FUNCTION_BLOCK PLCopenCallGroup IMPLEMENTS IPLCopenCall
VAR_INPUT
END_VAR
VAR_OUTPUT
END_VAR
VAR
    _callGroup : PLCopenCallGroupType;
END_VAR

// Copyright (c) 2024 Loupe (https://loupe.team), provided under the MIT License.

METHOD Aborted : BOOL
// Copyright (c) 2024 Loupe (https://loupe.team), provided under the MIT License.

_callGroup._syncAbort := TRUE;
END_METHOD

METHOD PRIVATE CheckStatus : BOOL
VAR
    _commandIndex : INT;
    _anyAbort : BOOL;
    _anyBusy : BOOL;
    _anyError : BOOL;
END_VAR
// Copyright (c) 2024 Loupe (https://loupe.team), provided under the MIT License.

//If it's not in the list
FOR _commandIndex := 0 TO GVLTcCommando.MAX_RELATED_GROUPS DO
    IF _callGroup._commands[_commandIndex].Command <> 0 THEN
        _callGroup._commands[_commandIndex]();

        IF _callGroup._commands[_commandIndex].CommandAborted THEN
            _anyAbort := TRUE;
        ELSIF _callGroup._commands[_commandIndex].Error THEN
            _anyError := TRUE;
        ELSIF _callGroup._commands[_commandIndex].Busy THEN
            _anyBusy := TRUE;
        ELSE
            _callGroup._commands[_commandIndex].Command := 0;
        END_IF
    END_IF
END_FOR

_callGroup._isError := FALSE;
_callGroup._isAbort := FALSE;
_callGroup._isDone := FALSE;

IF _anyError OR _callGroup._syncError THEN
    _callGroup._isError := TRUE;
ELSIF _anyAbort OR _callGroup._syncAbort THEN
    _callGroup._isAbort := TRUE;
ELSIF NOT _anyBusy THEN
    _callGroup._isDone := TRUE;
END_IF
END_METHOD

METHOD Errored : BOOL
VAR_INPUT
    ID : INT;
END_VAR
// Copyright (c) 2024 Loupe (https://loupe.team), provided under the MIT License.

_callGroup._syncError := TRUE;
END_METHOD

METHOD Finished : BOOL
// Copyright (c) 2024 Loupe (https://loupe.team), provided under the MIT License.

_callGroup._syncDone := TRUE;
END_METHOD

PROPERTY IsAbort : BOOL
GET
// Copyright (c) 2024 Loupe (https://loupe.team), provided under the MIT License.

CheckStatus();
IsAbort := _callGroup._isAbort;
END_GET
END_PROPERTY

PROPERTY IsDone : BOOL
GET
// Copyright (c) 2024 Loupe (https://loupe.team), provided under the MIT License.

CheckStatus();

//Check if we are done
IsDone := _callGroup._isDone;
END_GET
END_PROPERTY

PROPERTY IsError : BOOL
GET
// Copyright (c) 2024 Loupe (https://loupe.team), provided under the MIT License.

CheckStatus();

IsError := _callGroup._isError;
END_GET
END_PROPERTY

{warning 'add method implementation '}
METHOD PLCopenCall : PLCopenStatusBase
VAR_INPUT
    Command : IPLCopenCommand;
END_VAR
// Copyright (c) 2024 Loupe (https://loupe.team), provided under the MIT License.
END_METHOD

METHOD ResetCommands : BOOL
VAR
    _commandIndex : INT;
END_VAR
// Copyright (c) 2024 Loupe (https://loupe.team), provided under the MIT License.

//If it's not in the list
FOR _commandIndex := 0 TO GVLTcCommando.MAX_RELATED_GROUPS DO
    _callGroup._commands[_commandIndex].Clear();
END_FOR
END_METHOD

METHOD Start : BOOL
VAR_INPUT
    Command : IPLCopenCommand;
END_VAR
VAR
    _commandIndex : INT;
END_VAR
// Copyright (c) 2024 Loupe (https://loupe.team), provided under the MIT License.

// Check if it's already in the list
FOR _commandIndex := 0 TO GVLTcCommando.MAX_RELATED_GROUPS DO
    IF _callGroup._commands[_commandIndex].Command = Command THEN
        _callGroup._commands[_commandIndex].Exec(Command);
        Start := TRUE;
        RETURN;
    END_IF
END_FOR

// If it's not in the list
FOR _commandIndex := 0 TO GVLTcCommando.MAX_RELATED_GROUPS DO
    IF _callGroup._commands[_commandIndex].Command = 0 THEN
        _callGroup._commands[_commandIndex].Exec(Command);
        Start := TRUE;
        RETURN;
    END_IF
END_FOR

Start := FALSE;

//TODO: All out of commands.. Throw an error
END_METHOD

END_FUNCTION_BLOCK

(* stored: Version 1.1.0.1
   POU PLCopenCallGroup: Id {cba9c738-238a-4f8b-b4d1-3486de669f1d}, SpecialFunc None
   Folder PLCopenCaller: Id {b4b03af3-7533-4298-bf9d-09121bd9eae9}
   Method Aborted: Id {88516a3e-7cba-4182-ba66-c0dd75064666}
   Method CheckStatus: Id {69b5b758-9323-4002-906a-f59304b6dbf8}
   Method Errored: Id {2a110df0-07b9-4922-ba19-6e9f76e5caa7}
   Method Finished: Id {a2282568-2a57-49ba-abc9-a320ea291002}
   Property IsAbort: Id {96e569b0-457f-4c6e-bec1-643c895a8b9c}
   Get Get: Id {17cd4830-83fc-4522-8782-e508fda2b93d}
   Property IsDone: Id {c890f33c-6dc4-4031-a7ae-121d8a0f3c09}
   Get Get: Id {c8d0c1b7-b1e0-412a-9a10-7c15d2555f02}
   Property IsError: Id {28f1d1b2-fabc-44c9-968e-b0937bbe9074}
   Get Get: Id {24b146e6-8584-4378-a902-a6d936d8a944}
   Method PLCOpenCall: Id {e899a63b-d12d-476a-8450-473b6110f918}
   Method ResetCommands: Id {cd896665-6c8b-4e15-8c06-75a5a8e469f2}
   Method Start: Id {df0ebf2c-61b1-498a-bcc4-44d1e2466b24} *)
